// TIA Portal V21 export
TYPE "LAxisCtrl_typeTorqueLimiting"
TITLE = LAxisCtrl_typeTorqueLimiting
// Support: tech.team.motioncontrol@siemens.com
   STRUCT
      limit : LReal := -1.0;   // Value of force/torque limiting (in the configured unit of measurement) (Value >= 0.0: The specified value is used; Value < 0.0: Use of the default value configured in the technology object)
      mode : DInt := 0;   // 0: Force/Torque limiting; 1: Fixed stop detection
   END_STRUCT;
END_TYPE
